FUNCTION_BLOCK FB_ElectricityMeter_ABBA44213100
VAR_INPUT
	aElectricityMeterTelegramm	: ARRAY[1..cMBUS_MaxTelegrams] OF ST_MBus_Data2;
END_VAR
VAR_OUTPUT
	fWork : REAL; //Wh
	fPower : REAL; //W
END_VAR
VAR
	{attribute 'OPC.UA.DA' := '1'}
	sensorState : ST_ElectricityMeterState;
END_VAR

sensorState.fWork := STRING_TO_REAL(aElectricityMeterTelegramm[1].arrData[1].sValue);
sensorState.fPower := STRING_TO_REAL(aElectricityMeterTelegramm[2].arrData[2].sValue);

//set outputs
fWork := sensorState.fWork;
fPower := sensorState.fPower;

END_FUNCTION_BLOCK

(* stored: Version 1.1.0.1, ProductVersion 3.1.4024.10
   POU FB_ElectricityMeter_ABBA44213100: Id {3bc99379-6ea9-4c9b-ae55-3dca7b5d822b}, SpecialFunc None *)
